(* PLC project Blank Project, Blank Blank 1.0 *)
(* stored: creationDateTime 2016-05-18T21:14:07, modificationDateTime 2018-03-12T15:44:37 *)

PROGRAM My_Program
  VAR
    OnOff AT %QX0.0 : BOOL := 0;
    MaxGen AT %IW0 : INT := 300;
    CurrentGen AT %IW1 : INT := 200;
    ID AT %IW2 : INT := 5;
    TargetGen AT %QW0 : INT := 200;
  END_VAR
  VAR
    Delta : INT := 1;
    Increasing : BOOL := 0;
    Decreasing : BOOL := 0;
    Tick : BOOL := 0;
    Tick_Count : INT := 0;
    TON0 : TON;
  END_VAR
  VAR  (* added by the conversion: wires and edge detectors of the diagram *)
    R_TRIG1 : R_TRIG;
  END_VAR

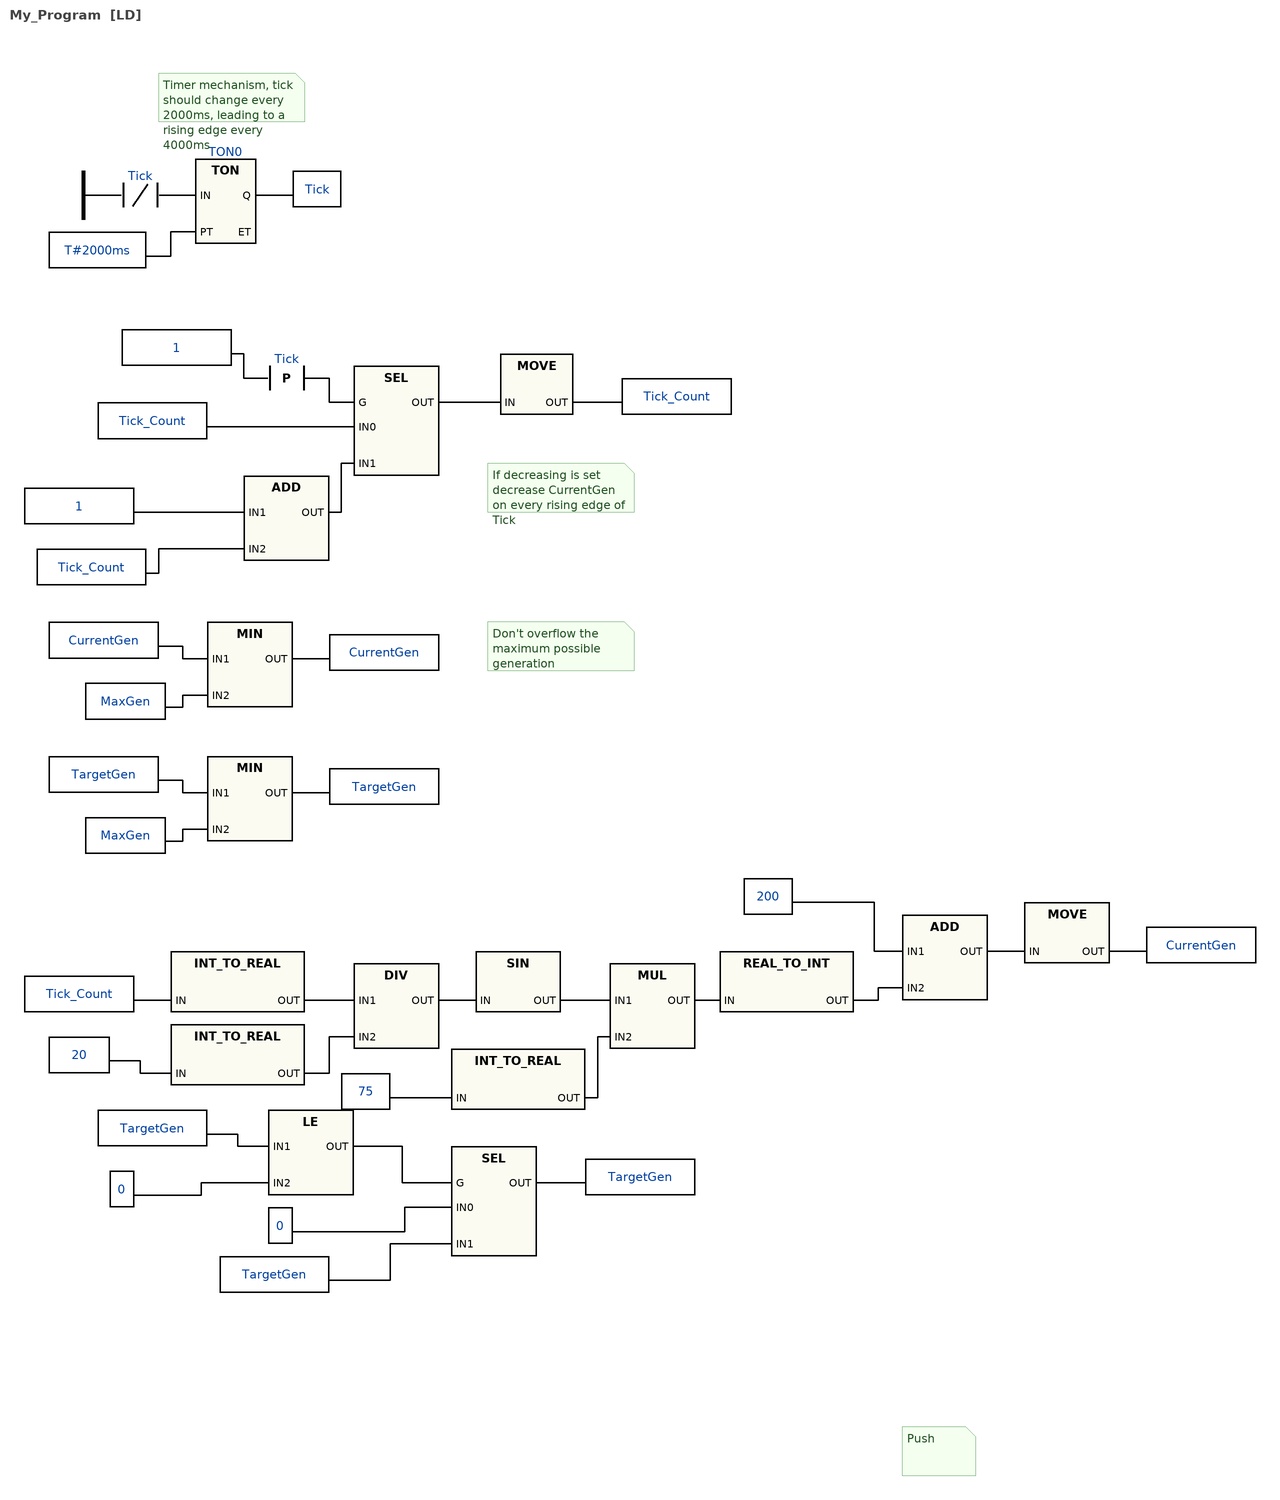
(* LD diagram, written out as Structured Text *)
(* Timer mechanism, tick should change every 2000ms, leading to a rising edge every 4000ms *)
TON0(IN := NOT Tick, PT := T#2000ms);
Tick := TON0.Q;
R_TRIG1(CLK := Tick);
Tick_Count := SEL(1 AND R_TRIG1.Q, Tick_Count, 1 + Tick_Count);
(* If decreasing is set decrease CurrentGen on every rising edge of Tick *)
(* Don't overflow the maximum possible generation *)
CurrentGen := MIN(CurrentGen, MaxGen);
TargetGen := MIN(TargetGen, MaxGen);
CurrentGen := 200 + REAL_TO_INT(SIN(INT_TO_REAL(Tick_Count) / INT_TO_REAL(20)) * INT_TO_REAL(75));
TargetGen := SEL(TargetGen <= 0, 0, TargetGen);
(* Push *)
END_PROGRAM

CONFIGURATION Config0
  RESOURCE Res0 ON PLC
    TASK TaskMain(INTERVAL := T#50ms, PRIORITY := 0);
    PROGRAM Inst0 WITH TaskMain : My_Program;
  END_RESOURCE
END_CONFIGURATION
